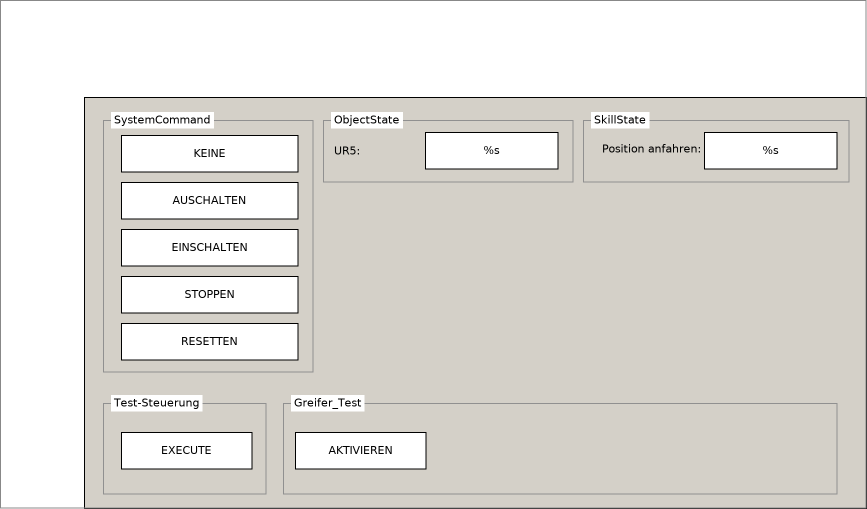
VISUALIZATION SystemState  // 867x509
    RoundedRectangle (84,97 783x412)
    GroupBox (103,112 210x260), "SystemCommand"
        RoundedRectangle (18,70 177x37), "AUSCHALTEN"
            OnMouseClick: execute { GVL.SystemCommand := 1; }
        RoundedRectangle (18,117 177x37), "EINSCHALTEN"
            OnMouseClick: execute { GVL.SystemCommand := 2; }
        RoundedRectangle (18,164 177x37), "STOPPEN"
            OnMouseClick: execute { GVL.SystemCommand := 3; }
        RoundedRectangle (18,211 177x37), "RESETTEN"
            OnMouseClick: execute { GVL.SystemCommand := 4; }
        RoundedRectangle (18,23 177x37), "KEINE"
            OnMouseClick: execute { GVL.SystemCommand := 0; }
    GroupBox (323,112 250x70), "ObjectState"
        RoundedRectangle (102,20 133x37), "%s", text variable: Anlage.UR5.P_State, input disabled if: TRUE
        Label (8,24 38x30), "UR5:"
    GroupBox (583,112 266x70), "SkillState"
        RoundedRectangle (121,20 133x37), "%s", text variable: MAIN.TestAblauf_1.P2P_Bewegung.P_State, input disabled if: TRUE
        Label (16,22 110x30), "Position anfahren:"
    GroupBox (103,395 163x99), "Test-Steuerung"
        RoundedRectangle (18,37 131x37), "EXECUTE"
            tap MAIN.Execute
    GroupBox (283,395 554x99), "Greifer_Test"
        RoundedRectangle (12,37 131x37), "AKTIVIEREN"
            OnMouseClick: execute { Anlage.Gripper.Aktivieren(); }
END_VISUALIZATION

(* stored: Version 1.1.0.1
   Visu SystemState: Id {61552118-6dd5-42b3-8f64-68d21c48a571} *)
